PROGRAM MAIN
VAR
END_VAR

END_PROGRAM

(* stored: Version 1.1.0.1
   POU MAIN: Id {18394bc5-d87f-4a2f-a4a2-2204f61f7f02} *)
